// TwinCAT 3 PLC project Analoog
// ProgramVersion: 3.1.4023.0
// libraries:
//   Tc2_Standard, * (Beckhoff Automation GmbH)
//   Tc2_System, * (Beckhoff Automation GmbH)
//   Tc3_Module, * (Beckhoff Automation GmbH)
// project tree:
//   / GlobalTextList.TcGTLO, PlcTask.TcTTO, Visualization Manager.TcVMO (not stored)
//   POUs/ CheckBounds.TcPOU, EX_02.TcPOU (not stored), EX_03.TcPOU (not stored), EX_04.TcPOU, EX_05.TcPOU, EX_06.TcPOU, EX_07.TcPOU, EX_08.TcPOU, EX_09.TcPOU, EX_10.TcPOU, EX_11.TcPOU (not stored), MAIN.TcPOU (not stored), EX_01.TcPOU, SCALING.TcPOU (not stored)
//   VISUs/ EX_01_V.TcVIS, EX_02_V.TcVIS, EX_03_V.TcVIS, EX_04_V.TcVIS, EX_05_V.TcVIS, EX_06_V.TcVIS, EX_07_V.TcVIS, EX_08_V.TcVIS, EX_09_V.TcVIS, EX_10_V.TcVIS, EX_11_V.TcVIS
// real-time tasks:
//   TASK PlcTask: cycle T#10ms, priority 20, ADS port 350

CONFIGURATION Analoog
    RESOURCE PLC ON TwinCAT3
        TASK PlcTask(INTERVAL := T#10ms, PRIORITY := 20);
        PROGRAM MAIN WITH PlcTask : MAIN;
    END_RESOURCE
END_CONFIGURATION

// ---- POUs/CheckBounds.TcPOU
// Implicitly generated code : DO NOT EDIT
FUNCTION CheckBounds : DINT
VAR_INPUT
	index, lower, upper: DINT;
END_VAR

// Implicitly generated code : Only an Implementation suggestion
{noflow}
IF  index < lower THEN
	CheckBounds := lower;
ELSIF  index > upper THEN
	CheckBounds := upper;
ELSE  
	CheckBounds := index;
END_IF
{flow}

END_FUNCTION

// ---- POUs/EX_04.TcPOU
PROGRAM EX_04
VAR
	Toggler: TP;
	tijd: TOF;
	
	period : INT;
	duty : INT;
END_VAR

VAR_INPUT
	potentio_freq : INT;
	potentio_duty : INT;
END_VAR

VAR_OUTPUT
	LED: BOOL;
END_VAR

Toggler(IN:= NOT tijd.Q, Q => LED);
tijd(IN:= Toggler.Q);

period := SCALING(input:=potentio_freq, imin:= 0, imax:= 32767, omin:= 500, omax:= 10000);
duty := SCALING(input:=potentio_duty, imin:= 0, imax:= 32767, omin:= 0, omax:= 100);

Toggler.PT := INT_TO_TIME(period*duty/100);
tijd.PT := INT_TO_TIME(period*(100-duty)/100);

END_PROGRAM

// ---- POUs/EX_05.TcPOU
PROGRAM EX_05

VAR
	druk_ingesteld_1 : INT;
	druk_ingesteld_2 : INT;
	druk_ingesteld_3 : INT;
	
	temp_min_value_1 : INT;
	temp_min_value_2 : INT;
	
	debiet_min_value_1 : INT;
END_VAR

VAR_INPUT
	druk_1 : INT;
	druk_2 : INT;
	druk_3 : INT;
	
	temp_1 : INT;
	temp_2 : INT;
	
	debiet_1 : INT;
END_VAR

VAR_OUTPUT
	productieProces_LED : BOOL;
	alarm_LED : BOOL;
END_VAR

IF((druk_1 < druk_ingesteld_1) AND (druk_2 < druk_ingesteld_2)) OR ((druk_1 < druk_ingesteld_1) AND (druk_3 < druk_ingesteld_3)) OR ((druk_2 < druk_ingesteld_2) AND (druk_3 < druk_ingesteld_3))
	THEN IF (debiet_1 < debiet_min_value_1)
		 	THEN productieProces_LED := FALSE;
		 END_IF
		 IF ((temp_1 < temp_min_value_1) AND (temp_2 < temp_min_value_2))
			THEN alarm_LED := TRUE;
				 productieProces_LED := FALSE;
		 END_IF
ELSE
	productieProces_LED := TRUE;
	alarm_LED := FALSE;
END_IF

END_PROGRAM

// ---- POUs/EX_06.TcPOU
PROGRAM EX_06

VAR
	TEMP_ASK : INT;
	TEMP_LIVE : INT;
END_VAR

VAR_INPUT
	potentio_ask: INT;
	potentio_live: INT;
END_VAR

VAR_OUTPUT
	LED : BOOL;
END_VAR

TEMP_ASK := SCALING(input:=potentio_ask, imin:= 0, imax:= 32767, omin:= 0, omax:= 30);
TEMP_LIVE := SCALING(input:=potentio_live, imin:= 0, imax:= 32767, omin:= 0, omax:= 30);

IF (TEMP_LIVE <= (TEMP_ASK-2))
	THEN LED := TRUE;
ELSIF (TEMP_LIVE >= (TEMP_ASK+2))
	THEN LED := FALSE;
END_IF

END_PROGRAM

// ---- POUs/EX_07.TcPOU
PROGRAM EX_07

VAR
	Toggler: TP;
	tijd: TOF;
	
	NIVEAU : INT;
END_VAR

VAR_INPUT
	NIVEAU_SENSOR : INT;
END_VAR

VAR_OUTPUT
	pomp_1 : BOOL;
	pomp_2 : BOOL;
	pomp_3 : BOOL;
	
	ALARM_LED : BOOL;
END_VAR

Toggler(IN:= NOT tijd.Q, Q => ALARM_LED);
tijd(IN:= Toggler.Q);


NIVEAU := SCALING(input:=NIVEAU_SENSOR, imin:= 0, imax:= 32767, omin:= 0, omax:= 100);

IF(NIVEAU < 50)
	THEN pomp_1 := FALSE;
	     pomp_2 := FALSE;
		 pomp_3 := FALSE;
		 ALARM_LED := FALSE;
ELSIF(NIVEAU < 70)
	THEN pomp_1 := TRUE;
		 pomp_2 := TRUE;
		 pomp_3 := FALSE;
		 ALARM_LED := FALSE;
ELSIF(NIVEAU < 80)
	THEN pomp_3 := TRUE;
		 ALARM_LED := FALSE;
ELSIF(NIVEAU > 80)
	THEN Toggler.PT := tijd.PT := T#300MS;
END_IF

END_PROGRAM

// ---- POUs/EX_08.TcPOU
PROGRAM EX_08
VAR
	GEWICHT : INT;
	mengen: TOF;
	MENG_NU : BOOL;
	R_TRIG : R_TRIG;
END_VAR

VAR_INPUT
	BALANS : INT;
	EMPTY : BOOL;
END_VAR

VAR_OUTPUT
	STOF_A_DIS : BOOL;
	STOF_B_DIS : BOOL;
	STOF_C_DIS : BOOL;
END_VAR

GEWICHT := SCALING(input:=BALANS, imin:= 0, imax:= 32767, omin:= 0, omax:= 100);
R_TRIG(CLK := MENG_NU);
mengen(IN:=R_TRIG.Q, PT:= T#5000MS);

IF(GEWICHT < 50)
	THEN MENG_NU := FALSE; 
		 STOF_A_DIS := TRUE;
	     STOF_B_DIS := FALSE;
	     STOF_C_DIS := FALSE;
ELSIF(GEWICHT < 60)
	THEN STOF_A_DIS := FALSE;
		 STOF_B_DIS := TRUE;
ELSIF(GEWICHT = 60)
	THEN STOF_A_DIS := FALSE;
		 STOF_B_DIS := FALSE;
		 MENG_NU := TRUE;
ELSIF(GEWICHT < 100) 
	THEN MENG_NU := FALSE;
		 STOF_C_DIS := TRUE;
ELSIF(GEWICHT = 100)
	THEN MENG_NU := TRUE;
END_IF

IF EMPTY THEN 
	GEWICHT := 0;
	BALANS := 0;
	STOF_A_DIS := FALSE;
	STOF_B_DIS := FALSE;
	STOF_C_DIS := FALSE;
END_IF

END_PROGRAM

// ---- POUs/EX_09.TcPOU
PROGRAM EX_09
VAR
	Toggler: TP;
	tijd: TOF;
	
	VOLTAGE : BYTE;
END_VAR

VAR_INPUT
	potentio : INT;
END_VAR

VAR_OUTPUT
	LED_1 : BOOL;
	LED_2 : BOOL;
END_VAR

Toggler(IN:= NOT tijd.Q, Q => LED_1);
tijd(IN:= Toggler.Q );

VOLTAGE := INT_TO_BYTE(SCALING(input:=potentio, imin:= 0, imax:= 32767, omin:= 0, omax:= 8));

IF(VOLTAGE <= 2)
	THEN Toggler.PT := tijd.PT := T#1000MS;
		 LED_2 := FALSE;
ELSIF(VOLTAGE <= 4)
	THEN Toggler.PT := tijd.PT := T#500MS;
		 LED_2 := FALSE;
ELSIF(VOLTAGE <= 6)
	THEN Toggler.PT := tijd.PT := T#250MS;
	 	 LED_2 := FALSE;
ELSIF(VOLTAGE > 6)
	THEN Toggler.PT := tijd.PT := T#100MS;
		 LED_2 := NOT(LED_1);
END_IF

END_PROGRAM

// ---- POUs/EX_10.TcPOU
PROGRAM EX_10
VAR

END_VAR

VAR_INPUT
	potentio_2k : INT;
	potentio_3k : INT;
	potentio_5k : INT;
END_VAR

VAR_OUTPUT
	slider_2k : INT;
	slider_3k : INT;
	slider_5k : INT;
	slider_10k : INT;
END_VAR

slider_2k := potentio_2k;
slider_3k := potentio_3k;
slider_5k := potentio_5k;
slider_10k := potentio_2k + potentio_3k + potentio_5k;

END_PROGRAM

// ---- POUs/EX_01.TcPOU
PROGRAM EX_01

VAR
	output: BYTE;
END_VAR

VAR_INPUT
	potentiometer: INT;
END_VAR

VAR_OUTPUT
	LED_0: BOOL;
	LED_1: BOOL;
	LED_2: BOOL;
	LED_3: BOOL;
	LED_4: BOOL;
	LED_5: BOOL;
	LED_6: BOOL;
	LED_7: BOOL;
END_VAR

output := INT_TO_BYTE(SCALING(input:=potentiometer, imin:= 0, imax:= 32767, omin:= 0, omax:= 255));

LED_0 := output.0;	// LSB
LED_1 := output.1; 
LED_2 := output.2; 
LED_3 := output.3; 
LED_4 := output.4; 
LED_5 := output.5; 
LED_6 := output.6;
LED_7 := output.7;	// MSB

END_PROGRAM

// ---- GlobalTextList.TcGTLO
TEXTLIST GlobalTextList
  168 = 'debiet_1'
  32 = 'druk_1'
  357 = 'druk_2'
  246 = 'druk_3'
  362 = 'Duty Cycle'
  182 = 'Frequency'
  364 = 'GEVRAAGD'
  851 = 'kk'
  515 = 'LIVE TEMP'
  624 = 'temp_1'
  194 = 'temp_2'
END_TEXTLIST

// ---- VISUs/EX_01_V.TcVIS
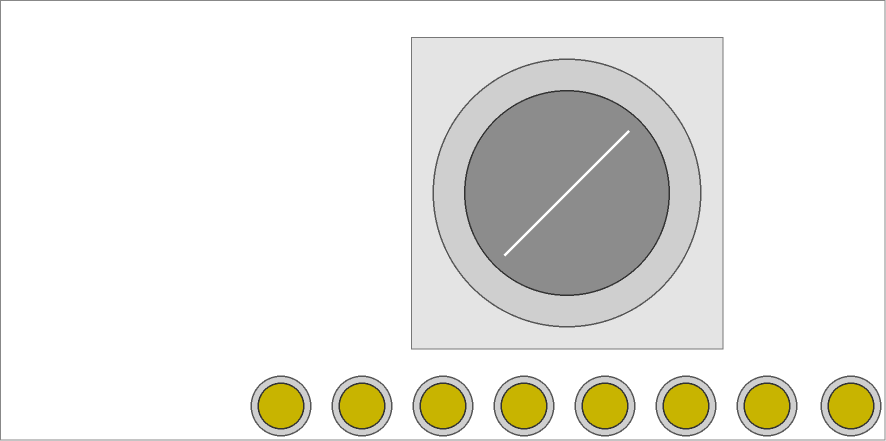
VISUALIZATION EX_01_V  // 886x441
    Lamp1 (732,371 70x70), variable: EX_01.LED_1, style: Lamp-Lamp1-Yellow
    Lamp1 (651,371 70x70), variable: EX_01.LED_2, style: Lamp-Lamp1-Yellow
    Lamp1 (246,371 70x70), variable: EX_01.LED_7, style: Lamp-Lamp1-Yellow
    Lamp1 (327,371 70x70), variable: EX_01.LED_6, style: Lamp-Lamp1-Yellow
    Lamp1 (408,371 70x70), variable: EX_01.LED_5, style: Lamp-Lamp1-Yellow
    Lamp1 (489,371 70x70), variable: EX_01.LED_4, style: Lamp-Lamp1-Yellow
    Lamp1 (570,371 70x70), variable: EX_01.LED_3, style: Lamp-Lamp1-Yellow
    Lamp1 (816,371 70x70), variable: EX_01.LED_0, style: Lamp-Lamp1-Yellow
    Potentiometer360 (353,37 428x312), variable: EX_01.potentiometer, style: Potentiometer-Potentiometer360-Gray, scale format: %.1f, scale 0..32760
        p2431819421: Outside
END_VISUALIZATION

// ---- VISUs/EX_02_V.TcVIS
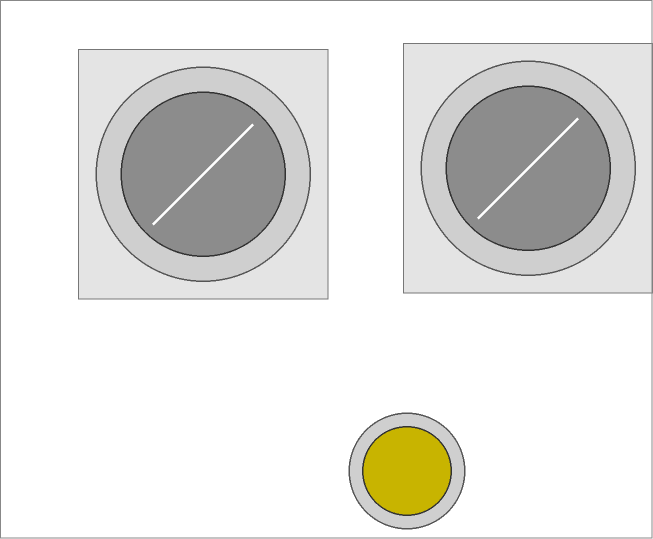
VISUALIZATION EX_02_V  // 653x539
    Potentiometer360 (78,49 250x250), variable: EX_02.potentiometer_ask, style: Potentiometer-Potentiometer360-Gray, scale format: %.1f, scale 0..32760
        p2431819421: Outside
    Potentiometer360 (403,43 250x250), variable: EX_02.potentiometer_live, style: Potentiometer-Potentiometer360-Gray, scale format: %.1f, scale 0..32760
        p2431819421: Outside
    Lamp1 (311,403 192x136), variable: EX_02.LED, style: Lamp-Lamp1-Yellow
END_VISUALIZATION

// ---- VISUs/EX_03_V.TcVIS
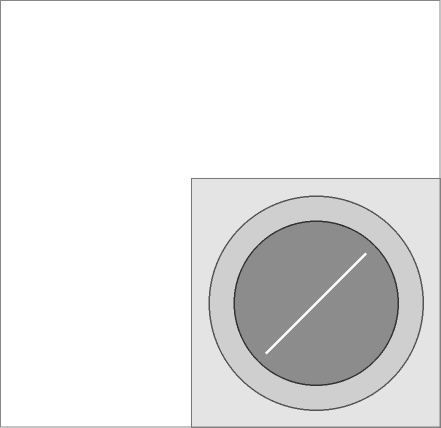
VISUALIZATION EX_03_V  // 441x428
    Potentiometer360 (191,178 250x250), variable: EX_03.potentiometer, style: Potentiometer-Potentiometer360-Gray, scale format: %.1f, scale 0..32760
        p2431819421: Outside
END_VISUALIZATION

// ---- VISUs/EX_04_V.TcVIS
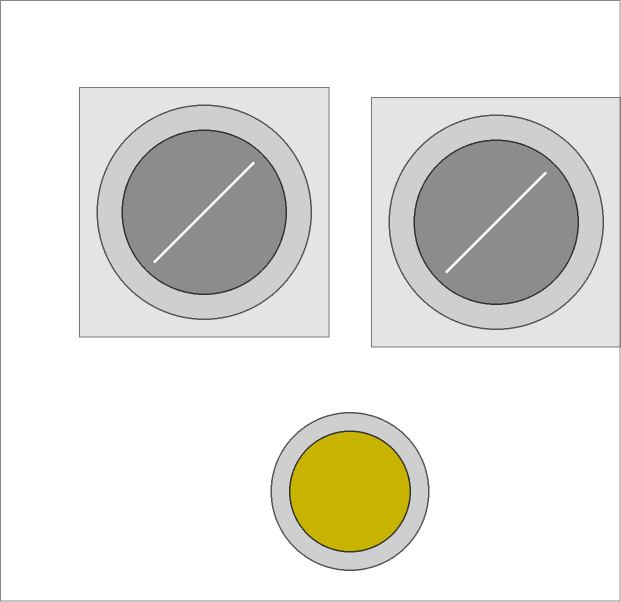
VISUALIZATION EX_04_V  // 621x602
    Potentiometer360 (79,87 250x250), variable: EX_04.potentio_freq, style: Potentiometer-Potentiometer360-Gray, scale format: %.1f, scale 0..32760
        p2431819421: Outside
        p518627256: Frequency
    Potentiometer360 (371,97 250x250), variable: EX_04.potentio_duty, style: Potentiometer-Potentiometer360-Gray, scale format: %.1f, scale 0..32760
        p2431819421: Outside
        p518627256: Duty Cycle
    Lamp1 (258,381 184x221), variable: EX_04.LED, style: Lamp-Lamp1-Yellow
END_VISUALIZATION

// ---- VISUs/EX_05_V.TcVIS
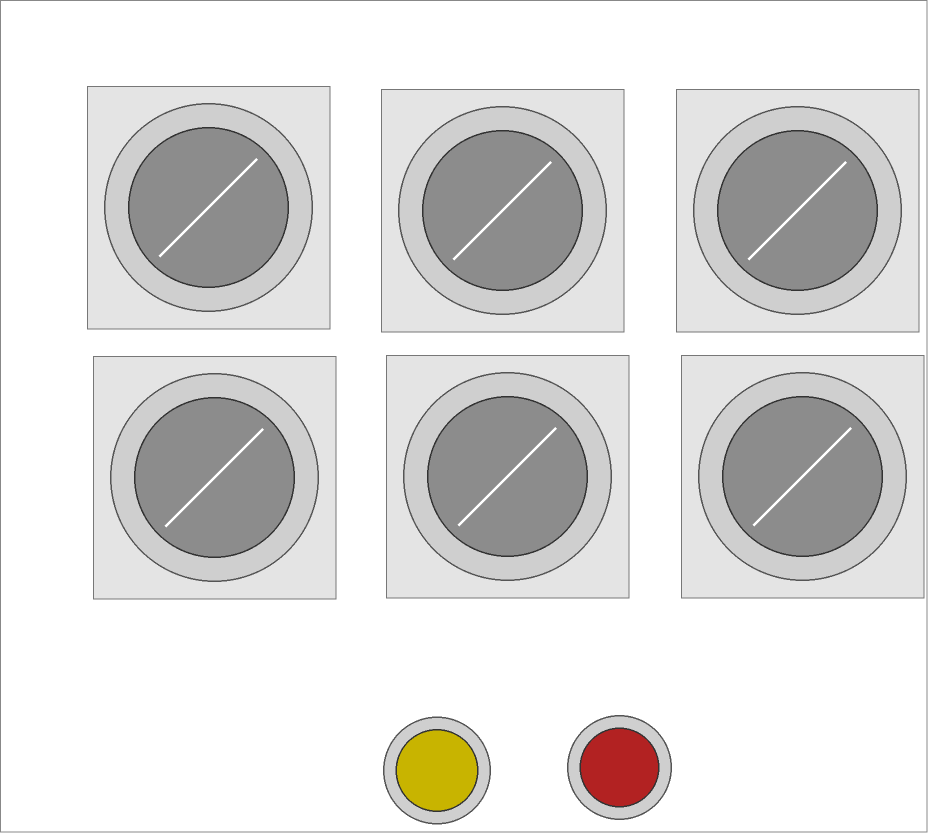
VISUALIZATION EX_05_V  // 928x833
    Potentiometer360 (89,356 251x243), variable: EX_05.temp_1, style: Potentiometer-Potentiometer360-Gray, scale format: %.1f, scale 0..32760
        p2431819421: Outside
        p518627256: temp_1
    Potentiometer360 (382,355 251x243), variable: EX_05.temp_2, style: Potentiometer-Potentiometer360-Gray, scale format: %.1f, scale 0..32760
        p2431819421: Outside
        p518627256: temp_2
    Potentiometer360 (677,355 251x243), variable: EX_05.debiet_1, style: Potentiometer-Potentiometer360-Gray, scale format: %.1f, scale 0..32760
        p2431819421: Outside
        p518627256: debiet_1
    Lamp1 (354,708 166x125), variable: EX_05.productieProces_LED, style: Lamp-Lamp1-Yellow
    Lamp1 (559,702 121x131), variable: EX_05.alarm_LED, style: Lamp-Lamp1-Red
    Potentiometer360 (83,86 251x243), variable: EX_05.druk_1, style: Potentiometer-Potentiometer360-Gray, scale format: %.1f, scale 0..32760
        p2431819421: Outside
        p518627256: druk_1
    Potentiometer360 (377,89 251x243), variable: EX_05.druk_2, style: Potentiometer-Potentiometer360-Gray, scale format: %.1f, scale 0..32760
        p2431819421: Outside
        p518627256: druk_2
    Potentiometer360 (672,89 251x243), variable: EX_05.druk_3, style: Potentiometer-Potentiometer360-Gray, scale format: %.1f, scale 0..32760
        p2431819421: Outside
        p518627256: druk_3
END_VISUALIZATION

// ---- VISUs/EX_06_V.TcVIS
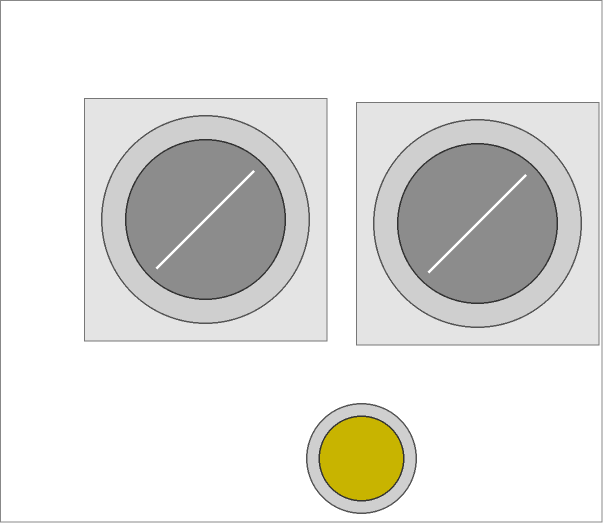
VISUALIZATION EX_06_V  // 603x523
    Potentiometer360 (80,98 251x243), variable: EX_06.potentio_ask, style: Potentiometer-Potentiometer360-Gray, scale format: %.1f, scale 0..32760
        p2431819421: Outside
    Potentiometer360 (352,102 251x243), variable: EX_06.potentio_live, style: Potentiometer-Potentiometer360-Gray, scale format: %.1f, scale 0..32760
        p2431819421: Outside
        p518627256: LIVE TEMP
    Lamp1 (280,394 163x129), variable: EX_06.LED, style: Lamp-Lamp1-Yellow
END_VISUALIZATION

// ---- VISUs/EX_07_V.TcVIS
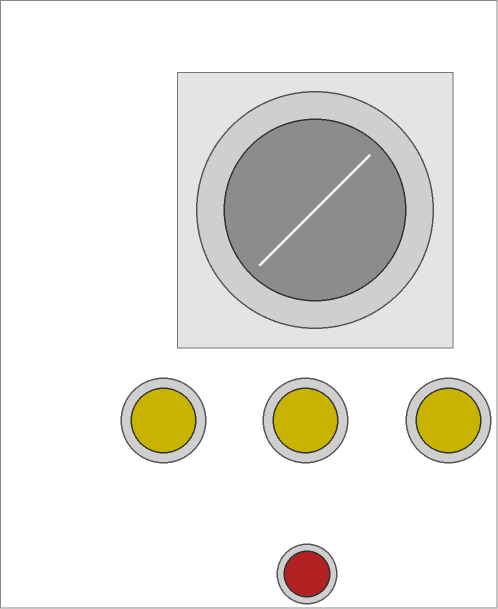
VISUALIZATION EX_07_V  // 498x609
    Potentiometer360 (158,72 314x276), variable: EX_07.NIVEAU_SENSOR, style: Potentiometer-Potentiometer360-Gray, scale format: %.1f, scale 0..32760
        p2431819421: Outside
    Lamp1 (114,369 99x103), variable: EX_07.pomp_1, style: Lamp-Lamp1-Yellow
    Lamp1 (272,539 70x70), variable: EX_07.ALARM_LED, style: Lamp-Lamp1-Red
    Lamp1 (256,369 99x103), variable: EX_07.pomp_2, style: Lamp-Lamp1-Yellow
    Lamp1 (399,369 99x103), variable: EX_07.pomp_3, style: Lamp-Lamp1-Yellow
END_VISUALIZATION

// ---- VISUs/EX_08_V.TcVIS
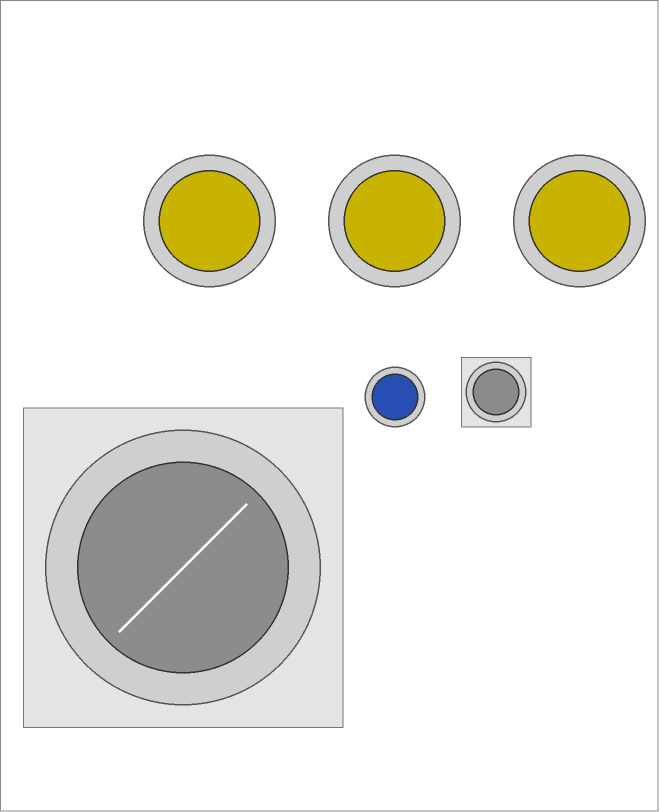
VISUALIZATION EX_08_V  // 659x812
    Lamp1 (130,144 159x154), variable: EX_08.STOF_A_DIS, style: Lamp-Lamp1-Yellow
    Lamp1 (315,144 159x154), variable: EX_08.STOF_B_DIS, style: Lamp-Lamp1-Yellow
    Lamp1 (500,144 159x154), variable: EX_08.STOF_C_DIS, style: Lamp-Lamp1-Yellow
    Lamp1 (360,362 70x70), variable: EX_08.mengen.Q, style: Lamp-Lamp1-Blue
    Potentiometer360 (23,323 320x489), variable: EX_08.BALANS, style: Potentiometer-Potentiometer360-Gray, scale format: %.1f, scale 0..32760
        p2431819421: Outside
    PushSwitch (461,357 70x70), variable: EX_08.EMPTY, behaviour: TAP, style: Switch-PushSwitch-Gray
END_VISUALIZATION

// ---- VISUs/EX_09_V.TcVIS
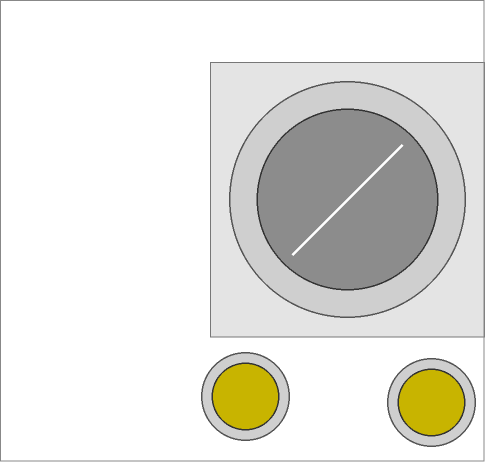
VISUALIZATION EX_09_V  // 485x462
    Potentiometer360 (210,55 275x289), variable: EX_09.potentio, style: Potentiometer-Potentiometer360-Gray, scale format: %.1f, scale 0..32670
        p2431819421: Outside
    Lamp1 (194,337 103x119), variable: EX_09.LED_1, style: Lamp-Lamp1-Yellow
    Lamp1 (380,343 103x119), variable: EX_09.LED_2, style: Lamp-Lamp1-Yellow
END_VISUALIZATION

// ---- VISUs/EX_10_V.TcVIS
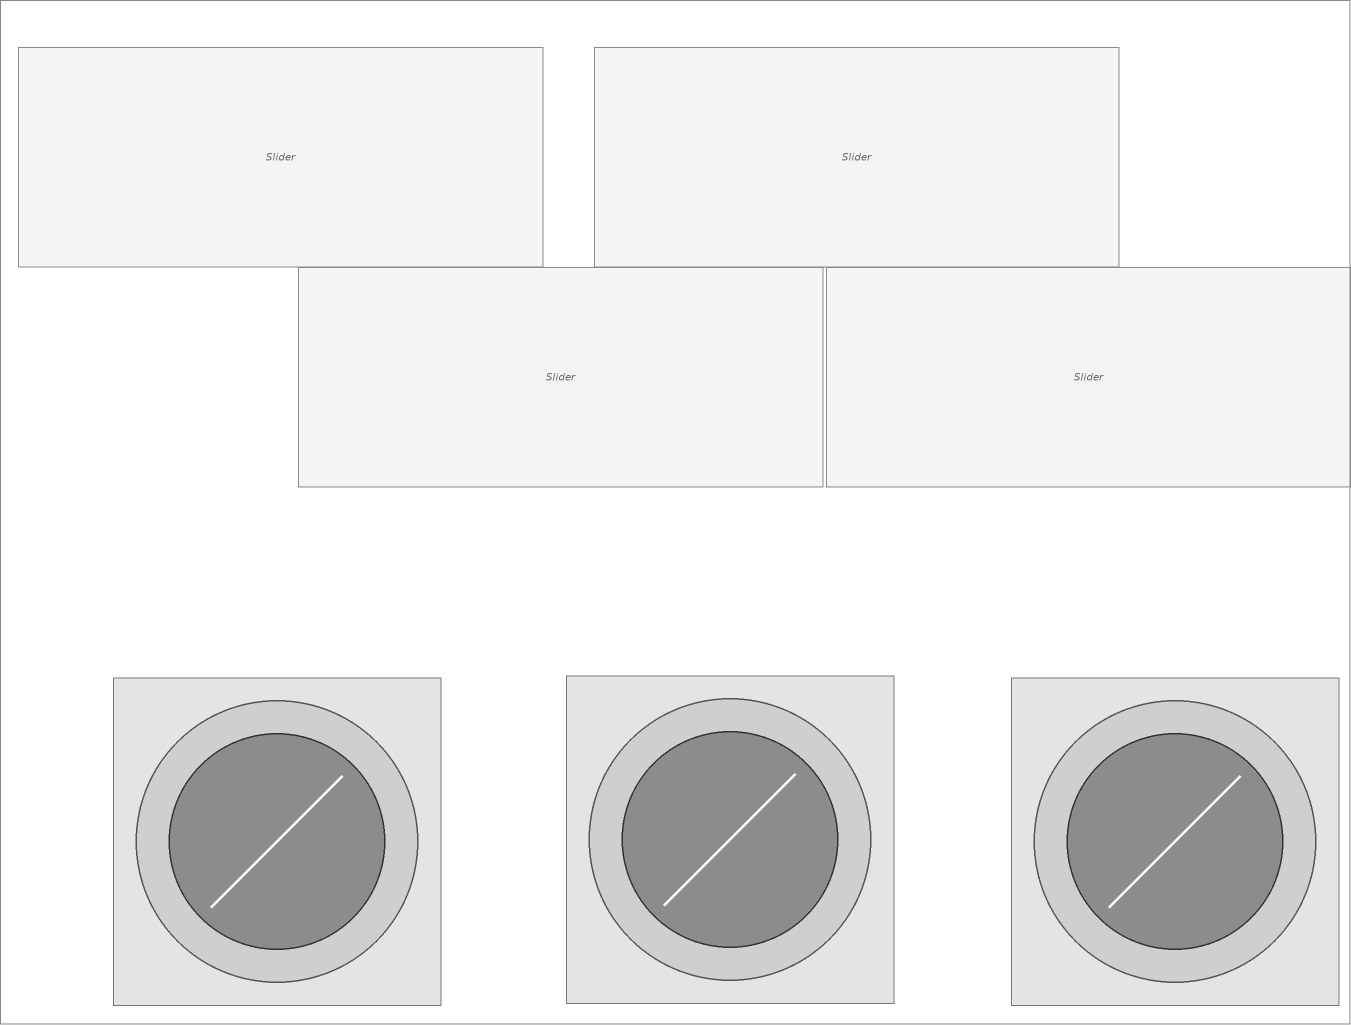
VISUALIZATION EX_10_V  // 1351x1025
    Slider (18,47 525x220), variable: EX_10.slider_2k, scale 0..2000
    Slider (298,267 525x220), variable: EX_10.potentio_5k, scale 0..5000
    Slider (594,47 525x220), variable: EX_10.potentio_3k, scale 0..3000
    Slider (826,267 525x220), variable: EX_10.slider_10k, scale 0..10000
    Potentiometer360 (1011,658 328x367), variable: EX_10.potentio_5k, style: Potentiometer-Potentiometer360-Gray, scale format: %.1f, scale 0..5000
        p2431819421: Outside
    Potentiometer360 (566,656 328x367), variable: EX_10.potentio_3k, style: Potentiometer-Potentiometer360-Gray, scale format: %.1f, scale 0..3000
        p2431819421: Outside
    Potentiometer360 (113,658 328x367), variable: EX_10.potentio_2k, style: Potentiometer-Potentiometer360-Gray, scale format: %.1f, scale 0..2000
        p2431819421: Outside
END_VISUALIZATION

// ---- VISUs/EX_11_V.TcVIS
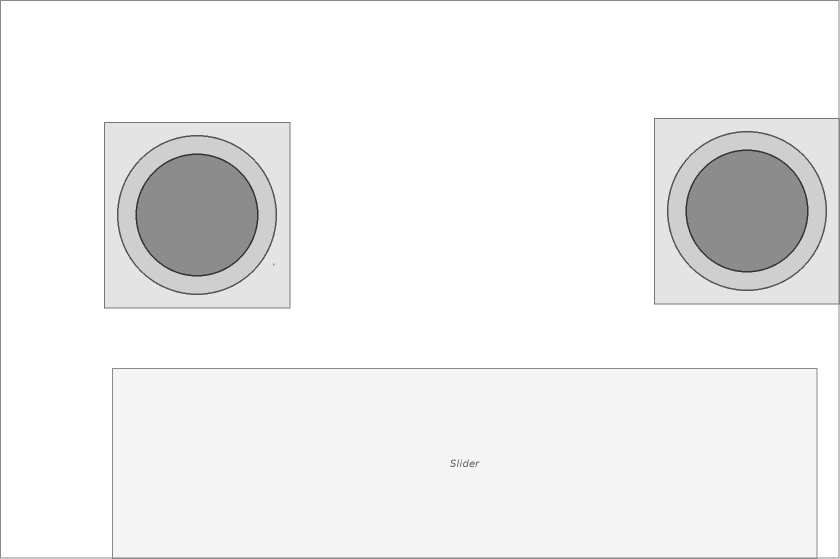
VISUALIZATION EX_11_V  // 840x559
    PushSwitch (104,115 186x200), variable: EX_11.bDown, behaviour: TAP, style: Switch-PushSwitch-Gray
    Slider (112,368 705x191), variable: EX_11.bVoltage, scale 0..10000
    Slider (273,264 1x0), scale 0..100
    PushSwitch (654,111 186x200), variable: EX_11.bUp, behaviour: TAP, style: Switch-PushSwitch-Gray
END_VISUALIZATION
